// TIA Portal V21 export
VAR_GLOBAL   // PLC tag table "K_Ricette"
END_VAR
VAR_GLOBAL CONSTANT   // user constants
   K_RicetteAdHmi : Int := 5;
   K_MacchinaARicetta_Spiedinatrice : Int := 2;
   K_MacchinaARicetta_Sterilizzatore : Int := 1;
END_VAR
